SUBAPPLICATION NVS_IN_AND_STORE_AIS (* NVS Laden und Speichern von AIS-Daten *)
  (* Standard: 61499-2; Description: Copyright (c) 2026 Meisterschulen am Ostbahnhof This program and the accompanying materials are made available under the terms of the Eclipse Public License 2.0 which is available at https://www.eclipse.org/legal/epl-2.0/ SPDX-License-Identifier: EPL-2.0 *)
  (* Version 1.0, 2026-04-24, Franz Höpfinger, Meisterschulen am Ostbahnhof, AIS adapter variant for String NVS storage with Subapp *)
  PACKAGE MyLib::sys;
  IMPORT isobus::UT::Q::const::IDs::ID_NULL;
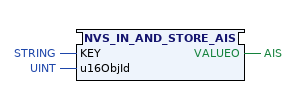
  VAR_INPUT
    KEY : STRING;
    u16ObjId : UINT := ID_NULL;
  END_VAR
  PLUGS
    VALUEO : adapter::types::unidirectional::AIS;
  END_PLUGS
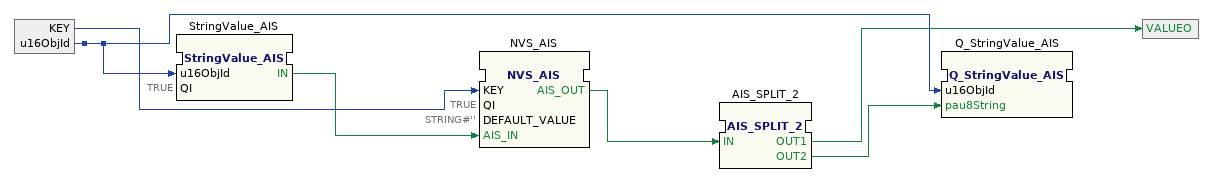
  FBS
    NVS_AIS : logiBUS::storage::esp32_nvs::NVS_AIS(QI := TRUE, DEFAULT_VALUE := STRING#'');
    StringValue_AIS : isobus::UT::io::StringValue::StringValue_AIS(QI := TRUE);
    Q_StringValue_AIS : isobus::UT::Q::Q_StringValue_AIS;
    AIS_SPLIT_2 : adapter::events::unidirectional::AIS_SPLIT_2;
  END_FBS
  DATA_CONNECTIONS
    u16ObjId TO Q_StringValue_AIS.u16ObjId;
    KEY TO NVS_AIS.KEY;
    u16ObjId TO StringValue_AIS.u16ObjId;
  END_CONNECTIONS
  ADAPTER_CONNECTIONS
    NVS_AIS.AIS_OUT TO AIS_SPLIT_2.IN;
    StringValue_AIS.IN TO NVS_AIS.AIS_IN;
    AIS_SPLIT_2.OUT1 TO VALUEO;
    AIS_SPLIT_2.OUT2 TO Q_StringValue_AIS.pau8String;
  END_CONNECTIONS
END_SUBAPPLICATION
